// TIA Portal V18 export
ORGANIZATION_BLOCK "01_OB1"   // OB1, LAD, ProgramCycle
TITLE = "Main Program Sweep (Cycle)"
{ S7_Optimized_Access := 'FALSE' }
AUTHOR : STD
FAMILY : System
VERSION : 2.0
// 系统程序段无需改动
// stored: AutoNumber false, SetENOAutomatically false
   VAR_TEMP
      OB1_EV_CLASS : Byte;   // Bits 0-3 = 1 (Coming event), Bits 4-7 = 1 (Event class 1)
      OB1_SCAN_1 : Byte;   // 1 (Cold restart scan 1 of OB 1), 3 (Scan 2-n of OB 1)
      OB1_PRIORITY : Byte;   // Priority of OB Execution
      OB1_OB_NUMBR : Byte;   // 1 (Organization block 1, OB1)
      OB1_RESERVED_1 : Byte;   // Reserved for system
      OB1_RESERVED_2 : Byte;   // Reserved for system
      OB1_PREV_CYCLE : Int;   // Cycle time of previous OB1 scan (milliseconds)
      OB1_MIN_CYCLE : Int;   // Minimum cycle time of OB1 (milliseconds)
      OB1_MAX_CYCLE : Int;   // Maximum cycle time of OB1 (milliseconds)
      OB1_DATE_TIME : Date_And_Time;   // Date and time OB1 started
      i : Int;
   END_VAR
   VAR_TEMP   // added for the SCL form of the ladder/FBD networks
      _w1 : Bool;
   END_VAR
BEGIN

REGION Network 1: Normal ON & OFF
   // 系统程序段
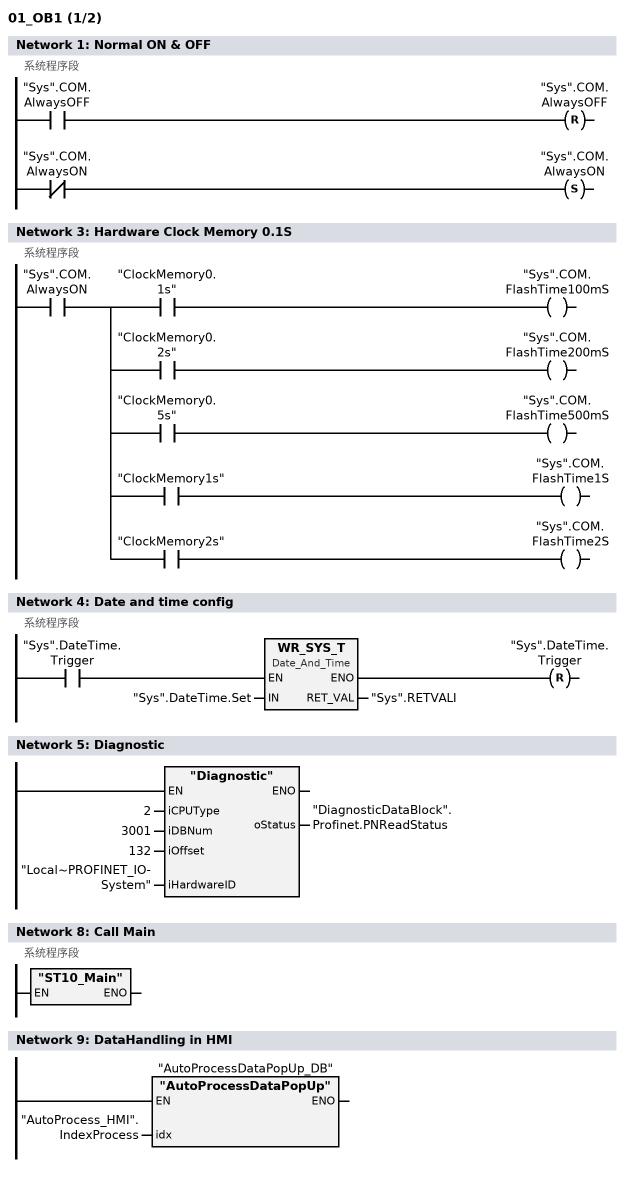
   RUNG wire#powerrail
      Contact( "Sys".COM.AlwaysOFF )
      R_Coil( "Sys".COM.AlwaysOFF )
   END_RUNG
   RUNG wire#powerrail
      I_Contact( "Sys".COM.AlwaysON )
      S_Coil( "Sys".COM.AlwaysON )
   END_RUNG
   // the same network as SCL:
   IF "Sys".COM.AlwaysOFF THEN "Sys".COM.AlwaysOFF := FALSE; END_IF;
   IF NOT "Sys".COM.AlwaysON THEN "Sys".COM.AlwaysON := TRUE; END_IF;
END_REGION

REGION Network 2 (SCL): ScanTime
   // System Function don't modify
   "Sys".ScanTime.CyclePrevious := #OB1_PREV_CYCLE;
   "Sys".ScanTime.CycleMin := #OB1_MIN_CYCLE;
   "Sys".ScanTime.CycleMax := #OB1_MAX_CYCLE;
END_REGION

REGION Network 3: Hardware Clock Memory 0.1S
   // 系统程序段
   RUNG wire#powerrail
      Contact( "Sys".COM.AlwaysON )
      wire#w1
      Contact( "ClockMemory0.1s" )
      Coil( "Sys".COM.FlashTime100mS )
   END_RUNG
   RUNG wire#w1
      Contact( "ClockMemory0.2s" )
      Coil( "Sys".COM.FlashTime200mS )
   END_RUNG
   RUNG wire#w1
      Contact( "ClockMemory0.5s" )
      Coil( "Sys".COM.FlashTime500mS )
   END_RUNG
   RUNG wire#w1
      Contact( "ClockMemory1s" )
      Coil( "Sys".COM.FlashTime1S )
   END_RUNG
   RUNG wire#w1
      Contact( "ClockMemory2s" )
      Coil( "Sys".COM.FlashTime2S )
   END_RUNG
   // the same network as SCL:
   "Sys".COM.FlashTime100mS := "Sys".COM.AlwaysON AND "ClockMemory0.1s";
   "Sys".COM.FlashTime200mS := "Sys".COM.AlwaysON AND "ClockMemory0.2s";
   "Sys".COM.FlashTime500mS := "Sys".COM.AlwaysON AND "ClockMemory0.5s";
   "Sys".COM.FlashTime1S := "Sys".COM.AlwaysON AND "ClockMemory1s";
   "Sys".COM.FlashTime2S := "Sys".COM.AlwaysON AND "ClockMemory2s";
END_REGION

REGION Network 4: Date and time config
   // 系统程序段
   RUNG wire#powerrail
      Contact( "Sys".DateTime.Trigger )
      { S7_Templates := "date_type := Date_And_Time" } WR_SYS_T(IN := "Sys".DateTime.Set, RET_VAL => "Sys".RETVALI)
      R_Coil( "Sys".DateTime.Trigger )
   END_RUNG
   // the same network as SCL:
   "Sys".RETVALI := WR_SYS_T(EN := "Sys".DateTime.Trigger, IN := "Sys".DateTime.Set, ENO => #_w1);
   IF #_w1 THEN "Sys".DateTime.Trigger := FALSE; END_IF;
END_REGION

REGION Network 5: Diagnostic
   RUNG wire#powerrail
      "Diagnostic"(iCPUType := 2, iDBNum := 3001, iOffset := 132, iHardwareID := "Local~PROFINET_IO-System", oStatus => "DiagnosticDataBlock".Profinet.PNReadStatus)
   END_RUNG
   // the same network as SCL:
   "Diagnostic"(iCPUType := 2,
                iDBNum := 3001,
                iOffset := 132,
                iHardwareID := "Local~PROFINET_IO-System",
                oStatus => "DiagnosticDataBlock".Profinet.PNReadStatus);
END_REGION

REGION Network 6 (SCL): Win
       "ST10_GeneralData".HMI.Win.WinBullfer := 0;
       FOR #i := 1 TO 10 DO
           "ST10_GeneralData".HMI.Win.WinBullfer := "ST10_GeneralData".HMI.Win.WinBullfer + "ST10_GeneralData".HMI.Win."10x弹窗"[#i] * 11 +"ST10_GeneralData".HMI.Win."20x弹窗"[2] * 21 +"ST10_GeneralData".HMI.Win."30x弹窗"[#i] * 31 +"ST10_GeneralData".HMI.Win."40x弹窗"[#i] * 41;
       END_FOR;
       "ST10_GeneralData".HMI.Win.WinBullfer := ABS("ST10_GeneralData".HMI.Win.WinBullfer);
       "ST10_GeneralData".HMI.Win.TON[1](IN := "ST10_GeneralData".HMI.Win.Win <> "ST10_GeneralData".HMI.Win.WinBullfer,
                          PT := T#0.5S);
   IF "ST10_GeneralData".HMI.Win.TON[1].Q THEN
       "ST10_GeneralData".HMI.Win.Win := "ST10_GeneralData".HMI.Win.WinBullfer;
       END_IF;
END_REGION

REGION Network 7: MES_Shopworx
END_REGION

REGION Network 8: Call Main
   // 系统程序段
   RUNG wire#powerrail
      "ST10_Main"()
   END_RUNG
   // the same network as SCL:
   "ST10_Main"();
END_REGION

REGION Network 9: DataHandling in HMI
   RUNG wire#powerrail
      "AutoProcessDataPopUp_DB"(idx := "AutoProcess_HMI".IndexProcess)
   END_RUNG
   // the same network as SCL:
   "AutoProcessDataPopUp_DB"(idx := "AutoProcess_HMI".IndexProcess);   // "AutoProcessDataPopUp"
END_REGION

REGION Network 10: 上电初始化设备模式_手动模式 / Power-on Initialization Device Mode _ Manual mode
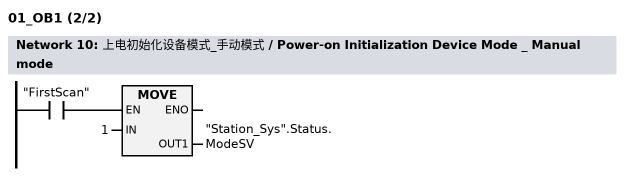
   RUNG wire#powerrail
      Contact( "FirstScan" )
      Move(in := 1, out1 => "Station_Sys".Status.ModeSV)
   END_RUNG
   // the same network as SCL:
   IF "FirstScan" THEN "Station_Sys".Status.ModeSV := 1; END_IF;
END_REGION
END_ORGANIZATION_BLOCK
